FUNCTION_BLOCK CylinderV (* Composite Function Block Type *)
  (* Standard: 61499-2 *)
  (* Version 0.0, 5/25/2016, Andrei, nxtControl GmbH, template *)
  PACKAGE Main;
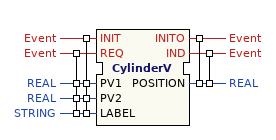
  EVENT_INPUT
    INIT WITH PV1, PV2, LABEL;
    REQ WITH PV1, PV2, LABEL; (* Normal Execution Request *)
  END_EVENT
  EVENT_OUTPUT
    INITO WITH POSITION; (* Initialization Confirm *)
    IND WITH POSITION; (* Execution Confirmation *)
  END_EVENT
  VAR_INPUT
    PV1 : REAL; (* Input event qualifier *)
    PV2 : REAL;
    LABEL : STRING;
  END_VAR
  VAR_OUTPUT
    POSITION : REAL; (* Output event qualifier *)
  END_VAR
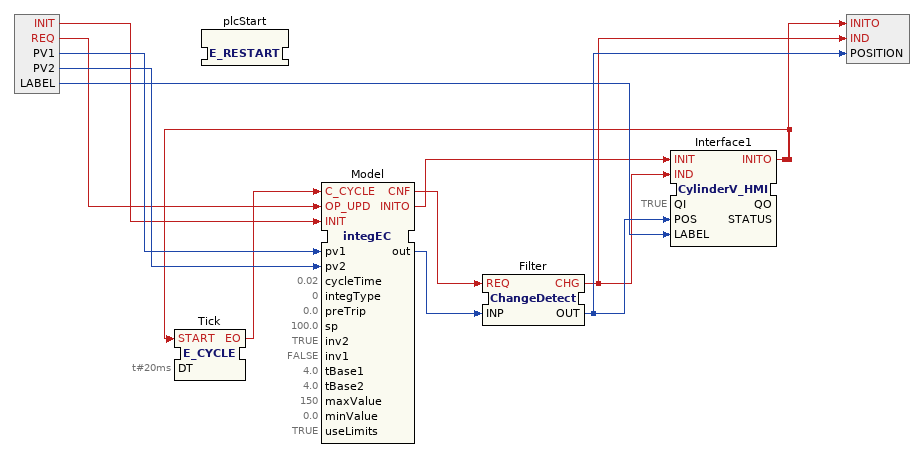
  FBS
    Tick : E_CYCLE(DT := t#20ms);
    Model : integEC(cycleTime := 0.02, integType := 0, preTrip := 0.0, sp := 100.0, inv2 := TRUE, inv1 := FALSE, tBase1 := 4.0, tBase2 := 4.0, maxValue := 150, minValue := 0.0, useLimits := TRUE);
    plcStart : E_RESTART;
    Interface1 : CylinderV_HMI(QI := TRUE);
    Filter : ChangeDetect;
  END_FBS
  EVENT_CONNECTIONS
    Tick.EO TO Model.C_CYCLE;
    Model.CNF TO Filter.REQ;
    REQ TO Model.OP_UPD;
    Filter.CHG TO IND;
    Model.INITO TO Interface1.INIT;
    Interface1.INITO TO INITO;
    Interface1.INITO TO Tick.START;
    Filter.CHG TO Interface1.IND;
    INIT TO Model.INIT;
  END_CONNECTIONS
  DATA_CONNECTIONS
    Model.out TO Filter.INP;
    PV1 TO Model.pv1;
    PV2 TO Model.pv2;
    Filter.OUT TO POSITION;
    Filter.OUT TO Interface1.POS;
    LABEL TO Interface1.LABEL;
  END_CONNECTIONS
END_FUNCTION_BLOCK
